// TIA Portal V20 export
DATA_BLOCK "DB_Recipe"   // DB5
{ S7_Optimized_Access := 'TRUE' }
// stored: MemoryReserve 100
   VAR
      Water_Fountain : String;
      Voltage : SInt;
      Min_Electrical_Current : UInt;
      Max_Electrical_Current : UInt;
      Time_End_Electrical_Current_Test : Time;
      Time_Start_Visual_Test : Time;
   END_VAR
BEGIN
END_DATA_BLOCK
